TYPE ST_Control :
STRUCT
	em8000: ST_ControlStewart;
	em1500: ST_ControlStewart;
	comau: ST_ControlComau;
	winch: ST_ControlWinch;
END_STRUCT
END_TYPE

(* stored: Version 1.1.0.1, ProductVersion 3.1.4026.8
   DUT ST_Control: Id {2b2e1f3a-3b90-4008-bd1d-0865302d3ba0} *)
